// TIA Portal V17 export
// export: Created 2023-04-20T08:24:45.7388178Z, ExportSetting WithDefaults, DisplayName Totally Integrated Automation Portal, DisplayVersion V17, DisplayName TIA Portal Openness, DisplayVersion V17, DisplayName TIA Portal Version Control Interface, DisplayVersion V17, DisplayName STEP 7 Professional, DisplayVersion V17, DisplayName STEP 7 Safety, DisplayVersion V17, DisplayName WinCC Advanced, DisplayVersion V17
ORGANIZATION_BLOCK "Main"   // OB1, LAD, ProgramCycle
TITLE = "Main Program Sweep (Cycle)"
{ S7_Optimized_Access := 'TRUE' }
VERSION : 0.1
// stored: AutoNumber true, IsIECCheckEnabled false, SetENOAutomatically false
   VAR_INPUT
      Initial_Call : Bool;   // Initial call of this OB
      Remanence : Bool;   // =True, if remanent data are available
   END_VAR
   VAR_TEMP
      Analog_value : Real;
   END_VAR
BEGIN

REGION Network 1
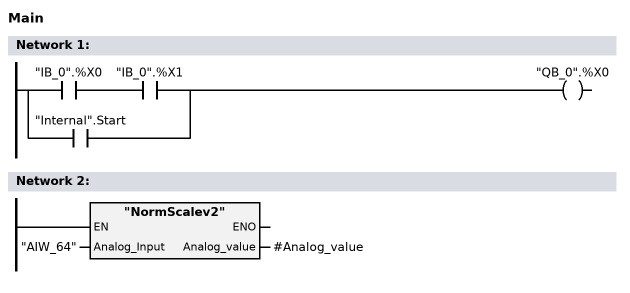
   RUNG wire#powerrail
      Contact( "IB_0".%X0 )
      Contact( "IB_0".%X1 )
      wire#w1
      Coil( "QB_0".%X0 )
   END_RUNG
   RUNG wire#powerrail
      Contact( "Internal".Start )
   END_RUNG wire#w1
   // the same network as SCL:
   "QB_0".%X0 := ("IB_0".%X0 AND "IB_0".%X1) OR "Internal".Start;
END_REGION

REGION Network 2
   RUNG wire#powerrail
      "NormScalev2"(Analog_Input := "AIW_64", Analog_value => #Analog_value)
   END_RUNG
   // the same network as SCL:
   "NormScalev2"(Analog_Input := "AIW_64", Analog_value => #Analog_value);
END_REGION
END_ORGANIZATION_BLOCK
